// TIA Portal V18 export
DATA_BLOCK "Comms_DB"   // DB22
// stored: AutoNumber false, InstanceOfName Comms, InstanceOfType FB
"Comms"
   // VAR
   //    DeviceLADDR : HW_IOSYSTEM;
   //    DeviceMode : UInt;
   //    DeviceReturn : Int;
   //    DeviceStates : Array[0..1023] of Bool;
   //    DeviceFault : Array[0..1023] of Bool;
   //    HpuPlcStatus : Bool;
   //    HpuPlcOnline : Bool;
   //    ConRIOStatus : Bool;
   //    ConRIOOnline : Bool;
   //    HpuHmiStatus : Bool;
   //    HpuHmiOnline : Bool;
   //    ConHmiStatus : Bool;
   //    ConHmiOnline : Bool;
   //    DHHmiStatus : Bool;
   //    DHHmiOnline : Bool;
   //    CouplerStatus : Bool;
   //    CouplerOnline : Bool;
   //    RemHearbeatOK : Bool;
   //    HBOn_TON { S7_SetPoint := 'True'} : TON_TIME;
   //    HeatbeatLost { S7_SetPoint := 'True'} : Bool;
   //    HBOff_TON { S7_SetPoint := 'True'} : TON_TIME;
   //    HBPosTrig : Bool;
   //    HBNegTrig : Bool;
   // END_VAR
BEGIN
END_DATA_BLOCK
